FUNCTION_BLOCK RpcServerConfigV1 Extends ServerConfigV1 IMPLEMENTS I_RpcServerConfig

PROPERTY PUBLIC HeaderKey_MethodName : T_MAXSTRING
GET
HeaderKey_MethodName := 'Method-Name';
END_GET
SET
// must keep so that it works with ANY
END_SET
END_PROPERTY

METHOD PUBLIC TryGetMethodNameFromRequest : BOOL
VAR_INPUT
	Request : I_Request;
	Destination : ANY;
END_VAR
TryGetMethodNameFromRequest := Request.Header.TryGetField(HeaderKey_MethodName,Destination);
END_METHOD

END_FUNCTION_BLOCK

(* stored: Version 1.1.0.1, ProductVersion 3.1.4024.12
   POU RpcServerConfigV1: Id {6a1246d9-7431-4d3e-91db-49877a54e466}, SpecialFunc None
   Folder Constants: Id {2881ef31-3af3-4535-82b6-167d7893e365}
   Property HeaderKey_MethodName: Id {1a5ae033-fd38-4b8d-97a6-154962797232}
   Get Get: Id {14a8f31e-ccaa-4e76-a81b-2dcd6b6bb2aa}
   Set Set: Id {c630eb4c-2924-4843-a93e-a295eb308278}
   Method TryGetMethodNameFromRequest: Id {421e7ac9-2f58-438a-bb83-66bee89f3edb} *)
